% RSLogix 500 project CTD QUE-1.RSS, saved by version 8.30.00.15 %
PROJECT "UNTITLED"    % processor: MicroLogix 1400 %

PROGRAM FILES
  LAD 2   4 rungs

DATA FILES
  O0 OUTPUT  6 elements
  I1 INPUT  8 elements
  S2 STATUS  66 elements
  B3 BINARY  1 elements
  T4 TIMER  1 elements
  C5 COUNTER  3 elements
  R6 CONTROL  1 elements
  N7 INTEGER  1 elements
  F8 FLOAT  1 elements

LADDER 2
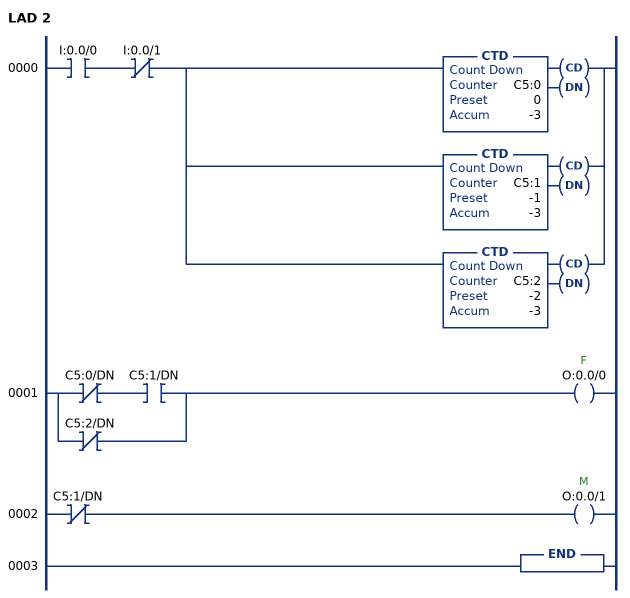
% Rung: 0 %
SOR XIC I:0.0/0 XIO I:0.0/1 BST CTD C5:0 0 -3 NXB BST CTD C5:1 -1 -3 NXB CTD C5:2 -2 -3 BND BND EOR
% Rung: 1 %
SOR BST XIO C5:0/DN XIC C5:1/DN NXB XIO C5:2/DN BND OTE O:0.0/0 EOR
%   O:0.0/0  F %
% Rung: 2 %
SOR XIO C5:1/DN OTE O:0.0/1 EOR
%   O:0.0/1  M %
% Rung: 3 %
SOR END EOR

DATA TABLE (non-zero values as saved)
DATA C5
% .PRE .ACC %
% C5:0 % 0 -3
% C5:1 % -1 -3
% C5:2 % -2 -3
